Fanuc KAREL source: kt00100.KL

-- PROVISIONAL review KL for V1013-1; original PC SHA256 d932cce1825f37957931f191757c2a1d7bf091280f12735a82093ff5fac3f1e6
-- Incomplete behavior may be omitted. Consult companion uncertainty JSON. Do not deploy.
PROGRAM KT00100
%NOLOCKGROUP
VAR
  I1 : INTEGER
  R2 : REAL
  OUT : REAL
BEGIN
  -- UNRESOLVED_PC offsets 5-16; opcodes 2E,23
  -- UNRESOLVED_PC offsets 21-32; opcodes 2E,23
  -- UNRESOLVED_PC offsets 37-59; opcodes 21,21,29,64,29,6C,23
  -- UNRESOLVED_PC offsets 64-68; opcodes 7F
END KT00100
